FUNCTION_BLOCK BOOL2BOOL
  {SET_ATTRIBUTE(OpcUa, SERVICE)}
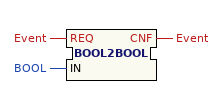
  EVENT_INPUT
    REQ;
  END_EVENT
  EVENT_OUTPUT
    CNF;
  END_EVENT
  VAR_INPUT
    IN : BOOL;
  END_VAR
END_FUNCTION_BLOCK
